RoboDK station: Sheet C - Top.rdk

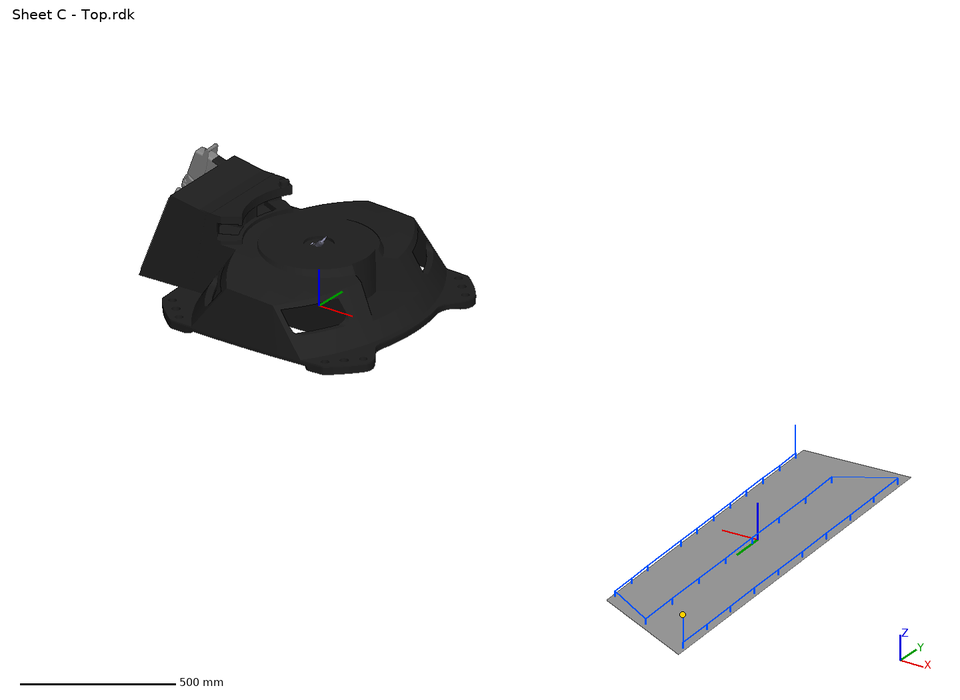
[picture v0: the station drawn from its stored meshes, robots at their saved joint values, targets as dots, program paths as lines]
Station Sheet C - Top (saved by RoboDK 5.2.3). Poses are relative to the parent item; angles as X-Y-Z fixed-axis rotations.
  - frame KUKA KR 210 R2700 extra Base at (0, 0, 0) mm
    - robot KUKA KR 210 R2700 extra: 6 axes, payload 210 kg, reach 2696 mm, repeatability 0.06 mm, weight 1068 kg
        joint limits [-185, -140, -120, -350, -125, -350] to [185, -5, 155, 350, 125, 350]; home [0, -90, 90, 0, 0, 0]; saved at [-26.436, -35.136, 121.604, -208.568, 35.866, 182.683]
      - tool Spindle, TCP at (32, 0, 260) mm, rotated rx 0 ry 39 rz 0 deg, size 157.3 x 72 x 259.9 mm
  - frame Frame 2 at (1698.49, 32.25, -372.68) mm, rotated rx 0 ry 0 rz -174.91 deg
    - object Sheet C - Top - box2 at (0, 0, 0) mm, size 400 x 1500 x 0.8 mm, geometry from Sheet C - Top - box2.stl
    - object Sheet C-box 2 Hole positioning - Top at (0, 0, 0) mm, 30 curves, geometry from Point 30
  - machining project Point settings: rotZ(0) | rotX(0)*rotY(0) | rotz(0) | onStart | onPathStart | onApproach | onPoint | onRetract | onFinish | SetRPM(%1) | SetTool(%1) | Extruder(%1) | default | default | OutOnMov(%1) | OutOffMov(%1) | onPathFinish | M_RunCode(%1)
  - program Point (156 instructions, listed below)
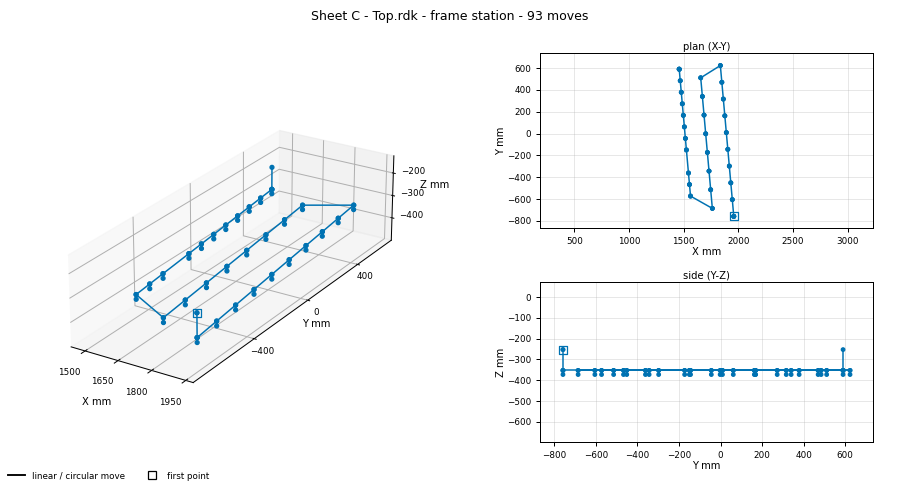
[picture p0: tool path of Sheet C - Top.rdk in frame station, 93 of 93 moves have a stored position in this frame; points joined in program order, loops and branches not executed]

--- program Point (robot KUKA KR 210 R2700 extra) ---
  Smooth(1)
  Set speed (1000.0 mm/s)
  Set Ref.: Frame 2
  Set Tool: Spindle
  Show Spindle
  MoveJ 1 to (-189, 810.01, 120) mm, rotated rx 180 ry 0 rz -5.09 deg; joints [24.221, -28.984, 92.88, -123.893, 18.121, 144.525]
  MoveL 2 to (-189, 810.01, 120) mm, rotated rx 180 ry 0 rz -5.09 deg; joints [24.221, -28.984, 92.88, -123.893, 18.121, 144.525]
  MoveL 3 to (-189, 810.01, 20) mm, rotated rx -180 ry 0 rz -5.09 deg; joints [24.221, -24.39, 90.434, -128.982, 19.398, 149.898]
  MoveL 4 to (-189, 810.01, 20) mm, rotated rx -180 ry 0 rz -5.09 deg; joints [24.221, -24.39, 90.434, -128.982, 19.398, 149.898]
  Set speed (50.0 mm/s)
  MoveL 5 to (-189, 810.01, 0) mm, rotated rx 180 ry 0 rz -5.09 deg; joints [24.221, -23.464, 89.895, -129.826, 19.644, 150.794]
  MoveL 6 to (-189, 810.01, 20) mm, rotated rx -180 ry 0 rz -5.09 deg; joints [24.221, -24.39, 90.434, -128.982, 19.398, 149.898]
  Set speed (1000.0 mm/s)
  MoveL 7 to (-189, 656.01, 20) mm, rotated rx -180 ry 0 rz -5.09 deg; joints [19.887, -25.619, 94.713, -142.155, 20.421, 159.643]
  Set speed (50.0 mm/s)
  MoveL 8 to (-189, 656.01, 0) mm, rotated rx 180 ry 0 rz -5.09 deg; joints [19.887, -24.669, 94.172, -142.817, 20.745, 160.35]
  MoveL 9 to (-189, 656.01, 20) mm, rotated rx -180 ry 0 rz -5.09 deg; joints [19.887, -25.619, 94.713, -142.155, 20.421, 159.643]
  Set speed (1000.0 mm/s)
  MoveL 10 to (-189, 502.01, 20) mm, rotated rx -180 ry 0 rz -5.09 deg; joints [15.224, -26.525, 98.192, -153.534, 21.766, 167.129]
  Set speed (50.0 mm/s)
  MoveL 11 to (-189, 502.01, 0) mm, rotated rx 180 ry 0 rz -5.09 deg; joints [15.224, -25.554, 97.645, -154.001, 22.147, 167.632]
  MoveL 12 to (-189, 502.01, 20) mm, rotated rx -180 ry 0 rz -5.09 deg; joints [15.224, -26.525, 98.192, -153.534, 21.766, 167.129]
  Set speed (1000.0 mm/s)
  MoveL 13 to (-189, 348.01, 20) mm, rotated rx -180 ry 0 rz -5.09 deg; joints [10.264, -27.161, 100.878, -163.415, 23.133, 172.694]
  Set speed (50.0 mm/s)
  MoveL 14 to (-189, 348.01, 0) mm, rotated rx 180 ry 0 rz -5.09 deg; joints [10.264, -26.171, 100.327, -163.703, 23.553, 173.007]
  MoveL 15 to (-189, 348.01, 20) mm, rotated rx -180 ry 0 rz -5.09 deg; joints [10.264, -27.161, 100.878, -163.415, 23.133, 172.694]
  Set speed (1000.0 mm/s)
  MoveL 16 to (-189, 194.01, 20) mm, rotated rx 180 ry 0 rz -5.09 deg; joints [5.057, -27.571, 102.773, -172.25, 24.289, 176.863]
  Set speed (50.0 mm/s)
  MoveL 17 to (-189, 194.01, 0) mm, rotated rx 180 ry 0 rz -5.09 deg; joints [5.057, -26.567, 102.217, -172.381, 24.734, 177.007]
  MoveL 18 to (-189, 194.01, 20) mm, rotated rx 180 ry 0 rz -5.09 deg; joints [5.057, -27.571, 102.773, -172.25, 24.289, 176.863]
  Set speed (1000.0 mm/s)
  MoveL 19 to (-189, 40.01, 20) mm, rotated rx -180 ry 0 rz -5.09 deg; joints [-0.325, -27.793, 103.871, -180.482, 25.078, 180.184]
  Set speed (50.0 mm/s)
  MoveL 20 to (-189, 40.01, 0) mm, rotated rx 180 ry 0 rz -5.09 deg; joints [-0.325, -26.78, 103.312, -180.474, 25.533, 180.176]
  MoveL 21 to (-189, 40.01, 20) mm, rotated rx -180 ry 0 rz -5.09 deg; joints [-0.325, -27.793, 103.871, -180.482, 25.078, 180.184]
  Set speed (1000.0 mm/s)
  MoveL 22 to (-189, -113.99, 20) mm, rotated rx 180 ry 0 rz -5.09 deg; joints [-5.792, -27.851, 104.169, -188.509, 25.42, 183.188]
  Set speed (50.0 mm/s)
  MoveL 23 to (-189, -113.99, 0) mm, rotated rx 180 ry 0 rz -5.09 deg; joints [-5.792, -26.836, 103.61, -188.369, 25.87, 183.033]
  MoveL 24 to (-189, -113.99, 20) mm, rotated rx 180 ry 0 rz -5.09 deg; joints [-5.792, -27.851, 104.169, -188.509, 25.42, 183.188]
  Set speed (1000.0 mm/s)
  MoveL 25 to (-189, -267.99, 20) mm, rotated rx -180 ry 0 rz -5.09 deg; joints [-11.246, -27.752, 103.665, -196.684, 25.31, 186.375]
  Set speed (50.0 mm/s)
  MoveL 26 to (-189, -267.99, 0) mm, rotated rx -180 ry 0 rz -5.09 deg; joints [-11.246, -26.741, 103.107, -196.413, 25.745, 186.075]
  MoveL 27 to (-189, -267.99, 20) mm, rotated rx -180 ry 0 rz -5.09 deg; joints [-11.246, -27.752, 103.665, -196.684, 25.31, 186.375]
  Set speed (1000.0 mm/s)
  MoveL 28 to (-189, -421.99, 20) mm, rotated rx 180 ry 0 rz -5.09 deg; joints [-16.591, -27.485, 102.362, -205.339, 24.827, 190.219]
  Set speed (50.0 mm/s)
  MoveL 29 to (-189, -421.99, 0) mm, rotated rx 180 ry 0 rz -5.09 deg; joints [-16.591, -26.484, 101.808, -204.933, 25.231, 189.771]
  MoveL 30 to (-189, -421.99, 20) mm, rotated rx 180 ry 0 rz -5.09 deg; joints [-16.591, -27.485, 102.362, -205.339, 24.827, 190.219]
  Set speed (1000.0 mm/s)
  MoveL 31 to (-189, -575.99, 20) mm, rotated rx 180 ry 0 rz -5.09 deg; joints [-21.741, -27.021, 100.264, -214.778, 24.122, 195.148]
  Set speed (50.0 mm/s)
  MoveL 32 to (-189, -575.99, 0) mm, rotated rx -180 ry 0 rz -5.09 deg; joints [-21.741, -26.035, 99.714, -214.232, 24.481, 194.548]
  MoveL 33 to (-189, -575.99, 20) mm, rotated rx 180 ry 0 rz -5.09 deg; joints [-21.741, -27.021, 100.264, -214.778, 24.122, 195.148]
  Set speed (1000.0 mm/s)
  MoveL 34 to (0, -480, 20) mm, rotated rx 180 ry 0 rz -5.09 deg; joints [-20.271, -28.948, 111.41, -204.281, 32.02, 184.917]
  Set speed (50.0 mm/s)
  MoveL 35 to (0, -480, 0) mm, rotated rx -180 ry 0 rz -5.09 deg; joints [-20.271, -27.869, 110.825, -203.962, 32.47, 184.539]
  MoveL 36 to (0, -480, 20) mm, rotated rx 180 ry 0 rz -5.09 deg; joints [-20.271, -28.948, 111.41, -204.281, 32.02, 184.917]
  Set speed (1000.0 mm/s)
  MoveL 37 to (0, -308.57, 20) mm, rotated rx 180 ry 0 rz -5.09 deg; joints [-13.663, -29.108, 113.188, -195.721, 33.273, 182.545]
  Set speed (50.0 mm/s)
  MoveL 38 to (0, -308.57, 0) mm, rotated rx 180 ry 0 rz -5.09 deg; joints [-13.663, -28.012, 112.595, -195.517, 33.757, 182.3]
  MoveL 39 to (0, -308.57, 20) mm, rotated rx 180 ry 0 rz -5.09 deg; joints [-13.663, -29.108, 113.188, -195.721, 33.273, 182.545]
  Set speed (1000.0 mm/s)
  MoveL 40 to (0, -137.14, 20) mm, rotated rx 180 ry 0 rz -5.09 deg; joints [-6.818, -29.162, 113.954, -187.711, 33.834, 181.109]
  Set speed (50.0 mm/s)
  MoveL 41 to (0, -137.14, 0) mm, rotated rx 180 ry 0 rz -5.09 deg; joints [-6.818, -28.058, 113.357, -187.611, 34.336, 180.988]
  MoveL 42 to (0, -137.14, 20) mm, rotated rx 180 ry 0 rz -5.09 deg; joints [-6.818, -29.162, 113.954, -187.711, 33.834, 181.109]
  Set speed (1000.0 mm/s)
  MoveL 43 to (0, 34.29, 20) mm, rotated rx 180 ry 0 rz -5.09 deg; joints [0.076, -29.145, 113.699, -179.913, 33.554, 179.987]
  Set speed (50.0 mm/s)
  MoveL 44 to (0, 34.29, 0) mm, rotated rx 180 ry 0 rz -5.09 deg; joints [0.076, -28.044, 113.104, -179.914, 34.06, 179.988]
  MoveL 45 to (0, 34.29, 20) mm, rotated rx 180 ry 0 rz -5.09 deg; joints [0.076, -29.145, 113.699, -179.913, 33.554, 179.987]
  Set speed (1000.0 mm/s)
  MoveL 46 to (0, 205.71, 20) mm, rotated rx 180 ry 0 rz -5.09 deg; joints [6.824, -29.045, 112.426, -171.986, 32.436, 178.537]
  Set speed (50.0 mm/s)
  MoveL 47 to (0, 205.71, 0) mm, rotated rx 180 ry 0 rz -5.09 deg; joints [6.824, -27.957, 111.837, -172.093, 32.93, 178.665]
  MoveL 48 to (0, 205.71, 20) mm, rotated rx 180 ry 0 rz -5.09 deg; joints [6.824, -29.045, 112.426, -171.986, 32.436, 178.537]
  Set speed (1000.0 mm/s)
  MoveL 49 to (0, 377.14, 20) mm, rotated rx -180 ry 0 rz -5.09 deg; joints [13.254, -28.805, 110.148, -163.548, 30.629, 176.116]
  Set speed (50.0 mm/s)
  MoveL 50 to (0, 377.14, 0) mm, rotated rx -180 ry 0 rz -5.09 deg; joints [13.254, -27.738, 109.569, -163.777, 31.096, 176.383]
  MoveL 51 to (0, 377.14, 20) mm, rotated rx -180 ry 0 rz -5.09 deg; joints [13.254, -28.805, 110.148, -163.548, 30.629, 176.116]
  Set speed (1000.0 mm/s)
  MoveL 52 to (0, 548.57, 20) mm, rotated rx 180 ry 0 rz -5.09 deg; joints [19.241, -28.337, 106.886, -154.151, 28.402, 172.094]
  Set speed (50.0 mm/s)
  MoveL 53 to (0, 548.57, 0) mm, rotated rx 180 ry 0 rz -5.09 deg; joints [19.241, -27.3, 106.319, -154.524, 28.825, 172.519]
  MoveL 54 to (0, 548.57, 20) mm, rotated rx 180 ry 0 rz -5.09 deg; joints [19.241, -28.337, 106.886, -154.151, 28.402, 172.094]
  Set speed (1000.0 mm/s)
  MoveL 55 to (0, 720, 20) mm, rotated rx -180 ry 0 rz -5.09 deg; joints [24.712, -27.547, 102.658, -143.289, 26.111, 165.873]
  Set speed (50.0 mm/s)
  MoveL 56 to (0, 720, 0) mm, rotated rx -180 ry 0 rz -5.09 deg; joints [24.712, -26.544, 102.103, -143.827, 26.471, 166.474]
  MoveL 57 to (0, 720, 20) mm, rotated rx -180 ry 0 rz -5.09 deg; joints [24.712, -27.547, 102.658, -143.289, 26.111, 165.873]
  Set speed (1000.0 mm/s)
  MoveL 58 to (189, 590.01, 20) mm, rotated rx 180 ry 0 rz -5.09 deg; joints [23.945, -29.198, 114.569, -153.423, 34.813, 176.711]
  Set speed (50.0 mm/s)
  MoveL 59 to (189, 590.01, 0) mm, rotated rx 180 ry 0 rz -5.09 deg; joints [23.945, -28.088, 113.969, -153.747, 35.269, 177.106]
  MoveL 60 to (189, 590.01, 20) mm, rotated rx 180 ry 0 rz -5.09 deg; joints [23.945, -29.198, 114.569, -153.423, 34.813, 176.711]
  Set speed (1000.0 mm/s)
  MoveL 61 to (189, 484.01, 20) mm, rotated rx -180 ry 0 rz -5.09 deg; joints [20.042, -29.27, 116.913, -158.894, 36.793, 178.651]
  Set speed (50.0 mm/s)
  MoveL 62 to (189, 484.01, 0) mm, rotated rx -180 ry 0 rz -5.09 deg; joints [20.042, -28.136, 116.3, -159.141, 37.28, 178.962]
  MoveL 63 to (189, 484.01, 20) mm, rotated rx -180 ry 0 rz -5.09 deg; joints [20.042, -29.27, 116.913, -158.894, 36.793, 178.651]
  Set speed (1000.0 mm/s)
  MoveL 64 to (189, 378.01, 20) mm, rotated rx -180 ry 0 rz -5.09 deg; joints [15.873, -29.246, 118.882, -164.003, 38.65, 179.841]
  Set speed (50.0 mm/s)
  MoveL 65 to (189, 378.01, 0) mm, rotated rx 180 ry 0 rz -5.09 deg; joints [15.873, -28.089, 118.257, -164.183, 39.161, 180.073]
  MoveL 66 to (189, 378.01, 20) mm, rotated rx -180 ry 0 rz -5.09 deg; joints [15.873, -29.246, 118.882, -164.003, 38.65, 179.841]
  Set speed (1000.0 mm/s)
  MoveL 67 to (189, 166.01, 20) mm, rotated rx 180 ry 0 rz -5.09 deg; joints [6.832, -29.055, 121.657, -173.524, 41.584, 180.466]
  Set speed (50.0 mm/s)
  MoveL 68 to (189, 166.01, 0) mm, rotated rx 180 ry 0 rz -5.09 deg; joints [6.832, -27.868, 121.013, -173.592, 42.125, 180.558]
  MoveL 69 to (189, 166.01, 20) mm, rotated rx 180 ry 0 rz -5.09 deg; joints [6.832, -29.055, 121.657, -173.524, 41.584, 180.466]
  Set speed (1000.0 mm/s)
  MoveL 70 to (189, 60.01, 20) mm, rotated rx 180 ry 0 rz -5.09 deg; joints [2.043, -28.963, 122.449, -178.096, 42.484, 180.184]
  Set speed (50.0 mm/s)
  MoveL 71 to (189, 60.01, 0) mm, rotated rx -180 ry 0 rz -5.09 deg; joints [2.043, -27.766, 121.799, -178.116, 43.031, 180.211]
  MoveL 72 to (189, 60.01, 20) mm, rotated rx 180 ry 0 rz -5.09 deg; joints [2.043, -28.963, 122.449, -178.096, 42.484, 180.184]
  Set speed (1000.0 mm/s)
  MoveL 73 to (189, -45.99, 20) mm, rotated rx 180 ry 0 rz -5.09 deg; joints [-2.848, -28.912, 122.837, -182.632, 42.921, 179.714]
  Set speed (50.0 mm/s)
  MoveL 74 to (189, -45.99, 0) mm, rotated rx 180 ry 0 rz -5.09 deg; joints [-2.848, -27.71, 122.184, -182.605, 43.469, 179.677]
  MoveL 75 to (189, -45.99, 20) mm, rotated rx 180 ry 0 rz -5.09 deg; joints [-2.848, -28.912, 122.837, -182.632, 42.921, 179.714]
  Set speed (1000.0 mm/s)
  MoveL 76 to (189, -151.99, 20) mm, rotated rx 180 ry 0 rz -5.09 deg; joints [-7.772, -28.914, 122.819, -187.186, 42.872, 179.224]
  Set speed (50.0 mm/s)
  MoveL 77 to (189, -151.99, 0) mm, rotated rx -180 ry 0 rz -5.09 deg; joints [-7.772, -27.713, 122.166, -187.113, 43.416, 179.125]
  MoveL 78 to (189, -151.99, 20) mm, rotated rx 180 ry 0 rz -5.09 deg; joints [-7.772, -28.914, 122.819, -187.186, 42.872, 179.224]
  Set speed (1000.0 mm/s)
  MoveL 79 to (189, -257.99, 20) mm, rotated rx 180 ry 0 rz -5.09 deg; joints [-12.656, -28.97, 122.394, -191.812, 42.347, 178.887]
  Set speed (50.0 mm/s)
  MoveL 80 to (189, -257.99, 0) mm, rotated rx 180 ry 0 rz -5.09 deg; joints [-12.656, -27.774, 121.745, -191.691, 42.882, 178.722]
  MoveL 81 to (189, -257.99, 20) mm, rotated rx 180 ry 0 rz -5.09 deg; joints [-12.656, -28.97, 122.394, -191.812, 42.347, 178.887]
  Set speed (1000.0 mm/s)
  MoveL 82 to (189, -363.99, 20) mm, rotated rx -180 ry 0 rz -5.09 deg; joints [-17.433, -29.065, 121.566, -196.567, 41.392, 178.867]
  Set speed (50.0 mm/s)
  MoveL 83 to (189, -363.99, 0) mm, rotated rx -180 ry 0 rz -5.09 deg; joints [-17.433, -27.878, 120.923, -196.394, 41.914, 178.635]
  MoveL 84 to (189, -363.99, 20) mm, rotated rx -180 ry 0 rz -5.09 deg; joints [-17.433, -29.065, 121.566, -196.567, 41.392, 178.867]
  Set speed (1000.0 mm/s)
  MoveL 85 to (189, -469.99, 20) mm, rotated rx -180 ry 0 rz -5.09 deg; joints [-22.042, -29.17, 120.34, -201.517, 40.086, 179.318]
  Set speed (50.0 mm/s)
  MoveL 86 to (189, -469.99, 0) mm, rotated rx 180 ry 0 rz -5.09 deg; joints [-22.042, -27.997, 119.705, -201.285, 40.587, 179.015]
  MoveL 87 to (189, -469.99, 20) mm, rotated rx -180 ry 0 rz -5.09 deg; joints [-22.042, -29.17, 120.34, -201.517, 40.086, 179.318]
  Set speed (1000.0 mm/s)
  MoveL 88 to (189, -575.99, 20) mm, rotated rx 180 ry 0 rz -5.09 deg; joints [-26.436, -29.251, 118.721, -206.731, 38.526, 180.379]
  Set speed (50.0 mm/s)
  MoveL 89 to (189, -575.99, 0) mm, rotated rx -180 ry 0 rz -5.09 deg; joints [-26.436, -28.096, 118.097, -206.436, 39, 180]
  MoveL 90 to (189, -575.99, 20) mm, rotated rx 180 ry 0 rz -5.09 deg; joints [-26.436, -29.251, 118.721, -206.731, 38.526, 180.379]
  MoveL 91 to (189, -575.99, 20) mm, rotated rx 180 ry 0 rz -5.09 deg; joints [-26.436, -29.251, 118.721, -206.731, 38.526, 180.379]
  Set speed (1000.0 mm/s)
  MoveL 92 to (189, -575.99, 20) mm, rotated rx 180 ry 0 rz -5.09 deg; joints [-26.436, -29.251, 118.721, -206.731, 38.526, 180.379]
  MoveL 93 to (189, -575.99, 120) mm, rotated rx 180 ry 0 rz -5.09 deg; joints [-26.436, -35.136, 121.604, -208.568, 35.866, 182.683]
